(* PLC project Tc2_Utilities.LrealIsNaN Demo, tc3-libraries-kb TwinCAT 3.1 *)
(* stored: creationDateTime 2026-05-10T11:00:00, modificationDateTime 2026-05-10T11:00:00 *)

PROGRAM P_Demo_LrealIsNaN
  VAR
    bResult : BOOL;  (* LrealIsNaN 的返回值 *)
    bRun : BOOL;  (* 触发一次调用 *)
    rX : LREAL;  (* 测试用本地变量 *)
  END_VAR

            // ============================================================
// Tc2_Utilities.LrealIsNaN 演示程序（FUNCTION）
// ============================================================
// 验证步骤：
//   1. 引用 Tc2_Utilities（及依赖类型所在的库）
//   2. 编译 + 登录
//   3. 强制 bRun := TRUE 一个周期
//   4. 观察 bResult 应为 FALSE（rX=3.14）
// ============================================================

rX := 3.14;
IF bRun THEN
    bResult := LrealIsNaN(rX);
    bRun := FALSE;
END_IF;

          
END_PROGRAM
